Staubli VAL3: run.pgx

public program run()
begin
  call taskPartMade()
  call IMMTiming()
end
